FUNCTION_BLOCK FB_MotionInterlocksSync EXTENDS FB_MotionInterlocks
VAR_INPUT
END_VAR
VAR_OUTPUT
END_VAR
VAR
    {attribute 'hide'}
    iMotionInterlocksShareData : I_MotionInterlocksShareData;
END_VAR

(*FB_Init is always available implicitly and it is used primarily for initialization.
The return value is not evaluated. For a specific influence, you can also declare the
methods explicitly and provide additional code there with the standard initialization
code. You can evaluate the return value.*)
METHOD FB_Init : BOOL
VAR_INPUT
    (* TRUE: the retain variables are initialized (reset warm / reset cold)*)
    bInitRetains	: BOOL;
    (* TRUE: the instance will be copied to the copy code afterward (online change)  *)
    bInCopyCode	: BOOL;
    iMotionLogger 		: I_MotionLogger;
    iMotionInterlocksShareData : I_MotionInterlocksShareData;
END_VAR
THIS^.iMotionInterlocksShareData := iMotionInterlocksShareData;
END_METHOD

END_FUNCTION_BLOCK

(* stored: Version 1.1.0.1
   POU FB_MotionInterlocksSync: Id {00f8072d-f625-44f2-84f3-5dd3d5c14806}, SpecialFunc None
   Method FB_Init: Id {f0be04ae-328f-4fac-8c99-e7ce1f739870} *)
